INTERFACE I_MutReceiverList EXTENDS Debug.I_Debug, I_ReceiverList

METHOD Extend 			: Results.Result
VAR_INPUT
	fbReceiverListExtend	: ReceiverListExtender;
END_VAR
END_METHOD

METHOD Push : Results.Result
VAR_INPUT
	iRec			: I_Receiver;
END_VAR
VAR_OUTPUT
	nPos			: UDINT;
END_VAR
END_METHOD

END_INTERFACE

(* stored: Version 1.1.0.1
   Itf I_MutReceiverList: Id {db452e49-1265-4060-8d55-6761eef6027a}
   Folder Push: Id {625f8185-241f-403c-b810-0092c3b60a0f}
   Method Extend: Id {c597d5d5-9ad4-400f-a8b3-25bbcf81c7c7}
   Method Push: Id {2ed16c57-2a93-4fdf-9c17-b7c00c671600} *)
